METHOD raiseError
VAR_INPUT
	bSetError : BOOL;
END_VAR
CASE iErrorId OF
	DOOR_DASHER_FAILED_TO_FIND_SOURCE_C_EYE_RISING_EDGE: 
		formatError('Failed to find source C-Eye rising edge', 'Turn Autofeed on and retry');
	DOOR_DASHER_FAILED_TO_FIND_SOURCE_D_EYE_RISING_EDGE: 
		formatError('Failed to find source D-Eye rising edge', 'Turn Autofeed on and retry');
	DOOR_DASHER_FAILED_TO_FIND_TARGET_C_EYE_RISING_EDGE: 
		formatError('Failed to find target C-Eye rising edge', 'Turn Autofeed on and retry');
	DOOR_DASHER_FAILED_TO_FIND_TARGET_D_EYE_RISING_EDGE: 
		formatError('Failed to find target D-Eye rising edge', 'Turn Autofeed on and retry');
	DOOR_DASHER_FAILED_TO_FIND_FALLING_EDGE_OF_TARGET_FEED_EYE_OR_RISING_EDGE_FENCE_EYE: 
		formatError('Failed to find falling edge of target feed eye or rising edge fence eye', 'Turn Autofeed on and retry');		
	DOOR_DASHER_TARGET_TRANSFER_TABLE_C_AND_D_FEED_EYES_MUST_BE_CLEAR: 
		formatError('Target transfer table C and D feed eyes must be clear', 'Turn Autofeed on and retry');
	DOOR_DASHER_FAILED_TO_FIND_SOURCE_A_EYE_RISING_EDGE: 
		formatError('Failed to find source A-Eye rising edge', 'Turn Autofeed on and retry');
	DOOR_DASHER_FAILED_TO_FIND_SOURCE_B_EYE_RISING_EDGE: 
		formatError('Failed to find source B-Eye rising edge', 'Turn Autofeed on and retry');
	DOOR_DASHER_FAILED_TO_FIND_TARGET_A_SIDE_EYE_RISING: 
		formatError('Failed to find target A-side eye rising edge', 'Turn Autofeed on and retry');
	DOOR_DASHER_FAILED_TO_FIND_TARGET_A_SIDE_EYE_FALLING: 
		formatError('Failed to find target A-side eye falling edge', 'Turn Autofeed on and retry');	
	DOOR_DASHER_FAILED_TO_FIND_TARGET_B_SIDE_EYE_RISING: 
		formatError('Failed to find target B-side eye rising edge', 'Turn Autofeed on and retry');
	DOOR_DASHER_FAILED_TO_FIND_TARGET_B_SIDE_EYE_FALLING: 
		formatError('Failed to find target B-side eye falling edge', 'Turn Autofeed on and retry');	
END_CASE
SUPER^.raiseError(bSetError);
END_METHOD

(* base implementation to record state calling history. 
 	Derrived FB's should override this method to replace the machine' specific type of eState *)
	
METHOD recordStateCallHistory
VAR_INPUT
	iState				: INT;
	iSubState			: INT;
END_VAR
VAR
	sCurTaskCycle 		: STRING;
    eState       		: E_DoorDasher_States; // todo: replace with the derrived STRUCT type (ie, E_HeadManager_States)
    eSubState			: E_SubState;
END_VAR
// DO NOT CHANGE BELOW!!!
// This was auto-generated by a Kval's UML tool.

sCurTaskCycle := TO_STRING(mainStateCallingData[iState, iSubState].nCycleIdFirstCall);
eState := iState;
eSubState := iSubState;

// Enter the state name into array
mainStateCallHistory[iStateCallHistoryIndex].sTaskCycle := sCurTaskCycle;
mainStateCallHistory[iStateCallHistoryIndex].sStateId := TO_STRING(iState);
mainStateCallHistory[iStateCallHistoryIndex].sStateDesc := TO_STRING(eState);
mainStateCallHistory[iStateCallHistoryIndex].sSubStateId := TO_STRING(iSubState);
mainStateCallHistory[iStateCallHistoryIndex].sSubStateDesc := TO_STRING(eSubState);

iStateCallHistoryIndex := iStateCallHistoryIndex + 1;
IF iStateCallHistoryIndex = MAX_STATE_CALL_HISTORY THEN
	iStateCallHistoryIndex := 0;
END_IF

// mark next index to record state call history
mainStateCallHistory[iStateCallHistoryIndex].sTaskCycle := '--';
mainStateCallHistory[iStateCallHistoryIndex].sStateId := '--';
mainStateCallHistory[iStateCallHistoryIndex].sStateDesc := '--';
mainStateCallHistory[iStateCallHistoryIndex].sSubStateId := '--';
mainStateCallHistory[iStateCallHistoryIndex].sSubStateDesc := '--';
END_METHOD

(* Any trigger that caused state transition (ie, cmd_bHome, cmd_bStartSequence, etc..) that
 	needs to be reset should go in here.
	 
	NOTE: The derived function block of KvalStateMachineBase_UmlSC should override/extend this method. *)
METHOD resetTriggers
SUPER ^.resetTriggers();
//TODO: reset all triggers (ie, cmd_bHome, cmd_bPark, etc...) here...
END_METHOD

METHOD setExternal
VAR 
	i : INT;
	tableIndex : INT;
END_VAR
FOR i:=iSourcePathIndex TO iTargetPathIndex DO
	tableIndex := stTargetPath.Path[i].TableIndex;
	MAIN.mainStateMachine.asmTableManagers[tableIndex].cmd_bExternal := TRUE;
END_FOR
END_METHOD

METHOD setInternal
VAR 
	i : INT;
	tableIndex : INT;
END_VAR
FOR i:=iSourcePathIndex TO iTargetPathIndex DO
	tableIndex := stTargetPath.Path[i].TableIndex;
	MAIN.mainStateMachine.asmTableManagers[tableIndex].cmd_bInternal := TRUE;
END_FOR
END_METHOD

METHOD setTargetDoorTrack
// transfer DoorTrack from source to target when done with transferring.
MAIN.mainStateMachine.asmTableManagers[cmd_iTarget].setDoorTrack(pstDoorTrack^);
END_METHOD

METHOD setTargetDoorTransferredInCompleted
MAIN.mainStateMachine.asmTableManagers[cmd_iTarget].setDoorTransferredInCompleted();
END_METHOD

METHOD sourceCrossFast
VAR 
	tableIndex : INT;
END_VAR
tableIndex := stTargetPath.Path[iSourcePathIndex].TableIndex;
MAIN.mainStateMachine.asmTableManagers[tableIndex].psmHcFeedMotor^.cmd_iSpeedRPM := MAIN.mainStateMachine.asmTableManagers[tableIndex].iCrossFeedFastSpeedRPM;
END_METHOD

METHOD sourceCrossFwd
VAR 
	tableIndex : INT;
END_VAR
tableIndex := stTargetPath.Path[iSourcePathIndex].TableIndex;
IF MAIN.mainStateMachine.asmTableManagers[tableIndex].config_bIsConveyorTable THEN
	MAIN.mainStateMachine.asmTableManagers[tableIndex].goFwd();
ELSE
	// inverted direction when crossing for the C234 feed.
	MAIN.mainStateMachine.asmTableManagers[tableIndex].goRev();
END_IF
END_METHOD

METHOD sourceCrossRev
VAR 
	tableIndex : INT;
END_VAR
tableIndex := stTargetPath.Path[iSourcePathIndex].TableIndex;
IF MAIN.mainStateMachine.asmTableManagers[tableIndex].config_bIsConveyorTable THEN
	MAIN.mainStateMachine.asmTableManagers[tableIndex].goRev();
ELSE
	// inverted direction when crossing for the C234 feed.
	MAIN.mainStateMachine.asmTableManagers[tableIndex].goFwd();
END_IF
END_METHOD

METHOD sourceGoFast
VAR 
	tableIndex : INT;
END_VAR
tableIndex := stTargetPath.Path[iSourcePathIndex].TableIndex;
MAIN.mainStateMachine.asmTableManagers[tableIndex].psmHcFeedMotor^.cmd_iSpeedRPM := MAIN.mainStateMachine.asmTableManagers[tableIndex].iFeedFastSpeedRPM;
END_METHOD

METHOD sourceGoFwd
VAR 
	tableIndex : INT;
END_VAR
tableIndex := stTargetPath.Path[iSourcePathIndex].TableIndex;
MAIN.mainStateMachine.asmTableManagers[tableIndex].goFwd();
END_METHOD

METHOD sourceGoRev
VAR 
	tableIndex : INT;
END_VAR
tableIndex := stTargetPath.Path[iSourcePathIndex].TableIndex;
MAIN.mainStateMachine.asmTableManagers[tableIndex].goRev();
END_METHOD

METHOD sourceStop
VAR 
	tableIndex : INT;
END_VAR
tableIndex := stTargetPath.Path[iSourcePathIndex].TableIndex;
MAIN.mainStateMachine.asmTableManagers[tableIndex].stop();
END_METHOD

METHOD stop
VAR 
	i : INT;
	
END_VAR
IF cmd_iSource <> cmd_iTarget THEN
	FOR i:=iSourcePathIndex TO iTargetPathIndex DO
		bStoppingSource := FALSE;
		bStoppingTarget := FALSE;
		iStopTableIndex := stTargetPath.Path[i].TableIndex;
		IF iStopTableIndex = cmd_iSource THEN
			// only stop the source if any of the following conditions is true...
			
			IF iSourceTrailingNeighborIndex = -1 THEN // no trailing neighbor
				bStoppingSource := TRUE;
			ELSE
				IF  // has trailing neighbor but it has no door 
					NOT MAIN.mainStateMachine.asmTableManagers[iSourceTrailingNeighborIndex].bHasDoor OR
					
					// has trailing neighbor but it has no door
					NOT (MAIN.mainStateMachine.asmTableManagers[iSourceTrailingNeighborIndex].smDoorDasher.bCrossTransferSeqRunning OR 
						MAIN.mainStateMachine.asmTableManagers[iSourceTrailingNeighborIndex].smDoorDasher.bInlineTransferSeqRunning) OR
						
					// trailing neighbor is transferring but not in the same direction as source's.
					stCurrentTargetNode.Direction <> eSourceTrailingNeighborNodeDirection
					THEN
					bStoppingSource := TRUE;
				END_IF
			END_IF
		ELSIF iStopTableIndex = cmd_iTarget THEN
			// always stop the target.
			bStoppingTarget := TRUE;
		END_IF
		IF bStoppingSource THEN
			MAIN.mainStateMachine.asmTableManagers[cmd_iSource].stop();			
		END_IF
		IF bStoppingTarget THEN
			MAIN.mainStateMachine.asmTableManagers[cmd_iTarget].stop();			
		END_IF
	END_FOR
END_IF
END_METHOD

METHOD targetCrossFast
VAR 
	tableIndex : INT;
END_VAR
tableIndex := stTargetPath.Path[iTargetPathIndex].TableIndex;
MAIN.mainStateMachine.asmTableManagers[tableIndex].psmHcFeedMotor^.cmd_iSpeedRPM := MAIN.mainStateMachine.asmTableManagers[tableIndex].iCrossFeedFastSpeedRPM;
END_METHOD

METHOD targetCrossFwd
VAR 
	tableIndex : INT;
END_VAR
tableIndex := stTargetPath.Path[iTargetPathIndex].TableIndex;
IF MAIN.mainStateMachine.asmTableManagers[tableIndex].config_bIsConveyorTable THEN
	MAIN.mainStateMachine.asmTableManagers[tableIndex].goFwd();
ELSE
	// inverted direction when crossing for the C234 feed.
	MAIN.mainStateMachine.asmTableManagers[tableIndex].goRev();
END_IF
END_METHOD

METHOD targetCrossRev
VAR 
	tableIndex : INT;
END_VAR
tableIndex := stTargetPath.Path[iTargetPathIndex].TableIndex;
IF MAIN.mainStateMachine.asmTableManagers[tableIndex].config_bIsConveyorTable THEN
	MAIN.mainStateMachine.asmTableManagers[tableIndex].goRev();
ELSE
	// inverted direction when crossing for the C234 feed.
	MAIN.mainStateMachine.asmTableManagers[tableIndex].goFwd();
END_IF
END_METHOD

METHOD targetCrossSlower
VAR 
	tableIndex : INT;
END_VAR
tableIndex := stTargetPath.Path[iTargetPathIndex].TableIndex;
MAIN.mainStateMachine.asmTableManagers[tableIndex].psmHcFeedMotor^.cmd_iSpeedRPM := MAIN.mainStateMachine.asmTableManagers[tableIndex].iCrossFeedSlowSpeedRPM/2;
END_METHOD

METHOD targetGoFast
VAR 
	tableIndex : INT;
END_VAR
tableIndex := stTargetPath.Path[iTargetPathIndex].TableIndex;
MAIN.mainStateMachine.asmTableManagers[tableIndex].psmHcFeedMotor^.cmd_iSpeedRPM := MAIN.mainStateMachine.asmTableManagers[tableIndex].iFeedFastSpeedRPM;
END_METHOD

METHOD targetGoFwd
VAR 
	tableIndex : INT;
END_VAR
tableIndex := stTargetPath.Path[iTargetPathIndex].TableIndex;
MAIN.mainStateMachine.asmTableManagers[tableIndex].goFwd();
END_METHOD

METHOD targetGoRev
VAR 
	tableIndex : INT;
END_VAR
tableIndex := stTargetPath.Path[iTargetPathIndex].TableIndex;
MAIN.mainStateMachine.asmTableManagers[tableIndex].goRev();
END_METHOD

METHOD targetStop
VAR 
	tableIndex : INT;
END_VAR
tableIndex := stTargetPath.Path[iTargetPathIndex].TableIndex;
MAIN.mainStateMachine.asmTableManagers[tableIndex].stop();
END_METHOD

METHOD updateSourceTargetDoorTrack
VAR_INPUT
END_VAR
setTargetDoorTrack();	
// is there new door-track data copied from the trailing door-dasher?
IF pstTable^.bDoorTrackDirty THEN
	pstTable^.bDoorTrackDirty := FALSE;
	pstTable^.stDoorTrack := pstTable^.stDoorTrackLast;
	pstTable^.setTableEmptyStatus(FALSE);
ELSE
	// clear source's DoorTrack.
	pstTable^.stDoorTrack := stDoorTrackDefault;
	pstTable^.setTableEmptyStatus(TRUE);					
END_IF
END_METHOD

(* Each transition has either or both a trigger (ie, cmd_bHome, cmd_bStartSequence, etc..)
	and a guard condition (i.e., bHeadReady AND bTableReady).
	This method updates all the state transitions.
	 
	NOTE: The derived function block of KvalStateMachineBase_UmlSC MUST override/extend this method. *)
METHOD updateStateTransitions
END_METHOD

END_FUNCTION_BLOCK

(* stored: Version 1.1.0.1, ProductVersion 3.1.4024.12
   POU SM_DoorDasher: Id {23c9881a-18b5-4abf-af0a-3e0dd6ea652d}, SpecialFunc None
   Folder uml: Id {a82803ea-1d13-4d35-992f-c60b15440d87}
   Method activateTablesCrossCyls: Id {05c75d4e-f7d8-4129-94ad-66490cc86be0}
   Method alignDoorAtTarget: Id {e6eeb860-7864-4324-8741-a95ab60a3f37}
   Method allTablesCrossCylsExtended: Id {d3933e58-8d86-4616-86ee-602741f84488}
   Method allTablesCrossCylsRetracted: Id {74919ebf-8554-4cdd-8005-be64ed63a915}
   Method allTablesExternal: Id {4de47f18-a166-47dc-aeee-f17521e728f0}
   Method allTablesMotorsMoving: Id {4656d3d1-7563-4c34-9233-25e8ebae783a}
   Method anyTableBusy: Id {63e4ab3c-caa3-4381-85dd-eb853db8eed6}
   Method anyTableExternal: Id {86dcb5db-2d73-446a-9594-c9b9072dd4cd}
   Method anyTableMotorMoving: Id {7fbf2b63-c87b-403d-8006-0e39f81545de}
   Method areTablesReady: Id {0f8d9675-aca7-4408-9451-2b112fd3d02d}
   Method centerDoorAtSource: Id {c2c58955-b2f9-4562-a5f9-b9fac23b7c8e}
   Method crossFast: Id {b6381d43-1785-4281-ba07-649ba972b00b}
   Method crossFwd: Id {2d0b5c36-61d6-45da-a596-3950000edb4e}
   Method crossRev: Id {7caff5ab-71e4-4b54-9559-4615e33252b3}
   Method crossSlow: Id {2c356925-3c51-4cc7-8665-01782da0295f}
   Method crossSlower: Id {12069367-42d2-4ec3-b95b-979bac03c5fa}
   Method crossTransferStart: Id {32918d41-538a-4201-aa69-0f6ef0c3998c}
   Method deactivateTablesCrossCyls: Id {7d02476d-a6e7-453a-874c-0e7c169cd4ba}
   Method doorDash: Id {d0189234-7e0e-45c1-bcd6-56803166cb1c}
   Method doState: Id {90b56b67-988a-4398-813b-266c6a3889a9}
   Method doState_UmlSC: Id {40c3d17d-657a-4d8e-af76-e3c339907801}
   Method feedinDoorAtTarget: Id {2697d187-c404-48b5-ade9-6f7007186497}
   Method findSourceLeadingNeighborTableIndex: Id {3c7cab24-48bf-4c0c-80fb-90b5cf81a0f3}
   Method findSourceTrailingNeighborTableIndex: Id {dec4e9b5-762f-4a71-9c04-6a90498c1d18}
   Method findTargetPathIndex: Id {666dcba6-c038-44f2-a7f0-7e385b1cf250}
   Method getStateDescription: Id {d62e3e46-7fa6-442f-af47-0f43e46466c3}
   Method getTableName: Id {1a362300-1194-41b5-809c-e76c2125118f}
   Method goFast: Id {43e26be5-9790-4965-8177-59396cfd0591}
   Method goFwd: Id {09b2cea7-6ab5-4ed3-adc1-08d18652be8f}
   Method goRev: Id {53396d2f-a5a3-4c1c-b252-c98352c1f119}
   Method goSlow: Id {9cf1f864-cdce-4bd3-b98d-0c131cde0809}
   Method initialize: Id {42e574aa-665f-46e4-94cc-e2c18b58dd9d}
   Method inlineTransferStart: Id {4325a22b-dc77-4bc5-873c-873090d7b1a4}
   Method isAligningDoorAtTarget: Id {7ddeca58-cf37-4adb-98fa-b0f17771e6e5}
   Method isAligningDoorAtTargetComplete: Id {3f5da155-c190-42a2-87ea-f4343c2b9a59}
   Method isFeedingInDoorAtTarget: Id {36f59534-59ab-4f74-8c2b-494ed014886b}
   Method isFeedingInDoorAtTargetComplete: Id {f6f874ce-e2c4-43c5-b34f-9a91699ad3fe}
   Method isSourceLeadingNeighborComplete: Id {06d85f6b-3b83-47f1-a365-539c88860708}
   Method isSourceLeadingNeighborReady: Id {ee07c25e-f095-4069-8bea-7c4fff07673e}
   Method isSourceMotorMoving: Id {ee24516f-3065-4bf7-83cb-d5b4659d9d2c}
   Method isSourceTableReady: Id {12c486f8-2b58-4cfa-a970-c38acf203ad7}
   Method isSourceTrailingNeighborComplete: Id {0ad6aae9-52f4-4a43-aec4-1abdd58064ea}
   Method isSourceTrailingNeighborReady: Id {7e212fc6-59f2-4241-8ef9-b3378694c22d}
   Method isTargetMotorMoving: Id {b686962a-2c71-45d8-95a7-1cb09e4103b2}
   Method isTargetTransferTableCandDsideDoorFeedEyesClear: Id {d65f8068-ebb2-4b62-882c-5d7f9e51c26f}
   Method postProcess: Id {f2a05d74-55a1-4aaa-b1e6-52218d61973e}
   Method preProcess: Id {d80ca6b5-b444-492c-a882-3774c8e2106b}
   Method raiseError: Id {16dab513-936b-40ca-912f-cd3e4323040f}
   Method recordStateCallHistory: Id {8167215a-9c5f-4707-9e8b-80558df34165}
   Method resetTriggers: Id {633220d9-2d6c-4393-bca7-87c6ccd1d8aa}
   Method setExternal: Id {db1c46ed-9e04-426a-8a59-0520fc6f85d6}
   Method setInternal: Id {352741f8-b989-49ae-b4d8-bcab00b07c19}
   Method setTargetDoorTrack: Id {f28b1093-5cd8-4fd4-bd82-5be5348fa789}
   Method setTargetDoorTransferredInCompleted: Id {0ea3f225-3ee8-4e07-b7fa-97f27db108e6}
   Method sourceCrossFast: Id {dd90b255-14d5-4d7e-8977-2f548c6fd542}
   Method sourceCrossFwd: Id {cc886053-d6ca-4d54-b227-99c9eea0c2be}
   Method sourceCrossRev: Id {69dd27bf-358a-4e05-afda-435c949e3b81}
   Method sourceGoFast: Id {f614ff2d-23e4-497d-a043-5ed80619d8f8}
   Method sourceGoFwd: Id {2b4bce7e-80bf-41b6-9cf9-40db612a63e9}
   Method sourceGoRev: Id {b63a1b85-1746-4927-b03a-9ad618730889}
   Method sourceStop: Id {87f17215-0eda-4704-b280-035358936c49}
   Method stop: Id {f8663887-c05e-4c8e-b2c2-a08da262ddab}
   Method targetCrossFast: Id {b9305575-cc0d-4fbc-a990-9c7de4792c19}
   Method targetCrossFwd: Id {91563f09-3bb6-493a-aa70-6a13e1a42386}
   Method targetCrossRev: Id {a6596fcb-798c-42bb-9eb1-5a1b5ad35e7f}
   Method targetCrossSlower: Id {9e93230e-3564-4cb4-a8d8-b4086fbeb724}
   Method targetGoFast: Id {7809e68b-e4d8-4416-a0bd-4418607a5855}
   Method targetGoFwd: Id {a515ec53-e03e-447e-b46e-5ba0079fdcdc}
   Method targetGoRev: Id {8c4893ec-6656-4e17-965d-02a3c5025400}
   Method targetStop: Id {1ce9c9e6-3ee2-41f1-aa05-da424fdfa0a5}
   Method updateSourceTargetDoorTrack: Id {19eaab80-dcc4-41f8-9fdc-97857fc39cd6}
   Method updateStateTransitions: Id {b1edd256-b9d3-452b-9249-3029129e0ffd} *)
